Fanuc KAREL source: kt00094.KL

-- PROVISIONAL review KL for V1013-1; original PC SHA256 b0e6494f6936e695342c2113397b159f648e8b532bf31456429b17daf141e060
-- Incomplete behavior may be omitted. Consult companion uncertainty JSON. Do not deploy.
PROGRAM KT00094
%NOLOCKGROUP
VAR
  OUT : REAL
-- UNRESOLVED_DECL H1 type=002017
-- UNRESOLVED_DECL Y2 type=002018
BEGIN
  -- UNRESOLVED_PC offsets 5-19; opcodes 2E,22,9D,33,B4
  -- UNRESOLVED_PC offsets 24-38; opcodes 2E,22,9D,33,B2
  -- UNRESOLVED_PC offsets 43-69; opcodes 22,9D,33,B3,22,9D,33,B1,54,64,23
  -- UNRESOLVED_PC offsets 74-78; opcodes 7F
END KT00094
